// Mitsubishi GX Works2 project: final1   PLC: FX3G

// global labels: Global1
VAR_GLOBAL
  dayOn AT Y000 : BOOL;
  endDay AT M2 : BOOL;
  dayOnn AT X007 : BOOL;
  emergncy AT X005 : BOOL;
  noInventory AT M1 : BOOL;
  dayBegin AT X007 : BOOL;
  sample AT X003 : BOOL;
  analogInput1 AT D8280 : INT;
  realInput AT D1200 : REAL;
END_VAR
VAR_GLOBAL CONSTANT
  const6 : REAL := 6.0;
  const5 : REAL := 5.0;
END_VAR
VAR_GLOBAL
  protein AT M3 : BOOL;
  regular AT M4 : BOOL;
END_VAR
VAR_GLOBAL CONSTANT
  proteinProteinPackageAmount : REAL := 320.0;
  honeytProteinPackageAmount : REAL := 160;
END_VAR
VAR_GLOBAL
  validProtein AT M31 : BOOL;
END_VAR
VAR_GLOBAL CONSTANT
  oatRegularPackageAmount : REAL := 400.0;
  proteinRegularPackageAmount : REAL := 160;
  honeyRegularPackageAmount : REAL := 120;
  honeyProteinPackageAmount : REAL := 160;
END_VAR
VAR_GLOBAL
  validRegular AT M41 : BOOL;
  mixTimer AT TC1 : BOOL;
END_VAR
VAR_GLOBAL CONSTANT
  const50 : INT := 50;
END_VAR
VAR_GLOBAL
  mixTimerOn AT TS1 : BOOL;
  MixLight AT Y003 : BOOL;
  try AT M20 : BOOL;
  oatContain AT D1300 : REAL;
  oatInput AT D1510 : REAL;
  honeyInput AT D1530 : REAL;
  honeyContein AT D1500 : REAL;
  proteinInput AT D1520 : REAL;
  proteinContein AT D1400 : REAL;
END_VAR
VAR_GLOBAL CONSTANT
  oatProteinPackageAmount : REAL := 240.0;
END_VAR
VAR_GLOBAL
  baking AT X002 : BOOL;
  bakeTimerRegular AT TC3 : BOOL;
  bakeTimerProtein AT TC2 : BOOL;
END_VAR
VAR_GLOBAL CONSTANT
  const40 : INT := 40;
END_VAR
VAR_GLOBAL
  bakeTimerProteinON AT TS2 : BOOL;
  bakeTimerRegularON AT TS3 : BOOL;
  flickerHelp AT M6 : BOOL;
  flicker1 AT TC4 : BOOL;
END_VAR
VAR_GLOBAL CONSTANT
  const10 : INT := 10;
END_VAR
VAR_GLOBAL
  flicerTimer1 AT TS4 : BOOL;
  flickerLight1 AT Y001 : BOOL;
  flicker2 AT TC5 : BOOL;
  flicerTimer2 AT TS5 : BOOL;
  flickerLight2 AT Y002 : BOOL;
  finishBake AT M5 : BOOL;
  packing AT X006 : BOOL;
  packingOneBar AT X000 : BOOL;
  countingOneBar AT CC0 : BOOL;
END_VAR
VAR_GLOBAL CONSTANT
  cont1 : INT := 1;
END_VAR
VAR_GLOBAL
  counting8bars AT CC1 : BOOL;
END_VAR
VAR_GLOBAL CONSTANT
  const8 : INT := 8;
END_VAR
VAR_GLOBAL
  counterStarter AT CS0 : BOOL;
  counterStopper AT CS1 : BOOL;
  packingLight AT Y004 : BOOL;
  packageFinished AT M7 : BOOL;
  logInput AT D1250 : REAL;
END_VAR
VAR_GLOBAL CONSTANT
  const400 : REAL := 400.0;
END_VAR
VAR_GLOBAL
  analogPackages AT D1260 : REAL;
  packegesOutput AT D8282 : INT;
END_VAR
VAR_GLOBAL CONSTANT
  const0 : REAL;
  const1 : REAL := 1.0;
END_VAR
VAR_GLOBAL
  totalPackeges AT D1600 : REAL;
  restartPackingCount AT CN1 : INT;
END_VAR
VAR_GLOBAL CONSTANT
  const40Float : REAL := 40.0;
END_VAR
VAR_GLOBAL
  test111 AT M99 : BOOL;
  test888 AT M99 : BOOL;
  noInventory2 AT M19 : BOOL;
END_VAR

// task Task_01 (event TRUE, interval 0, priority 31): POU_01

PROGRAM POU_01
(* structured ladder/FBD written out as ST: instructions are called as NAME(EN, inputs, outputs); _pN, _eN, _tN stand for wires *)
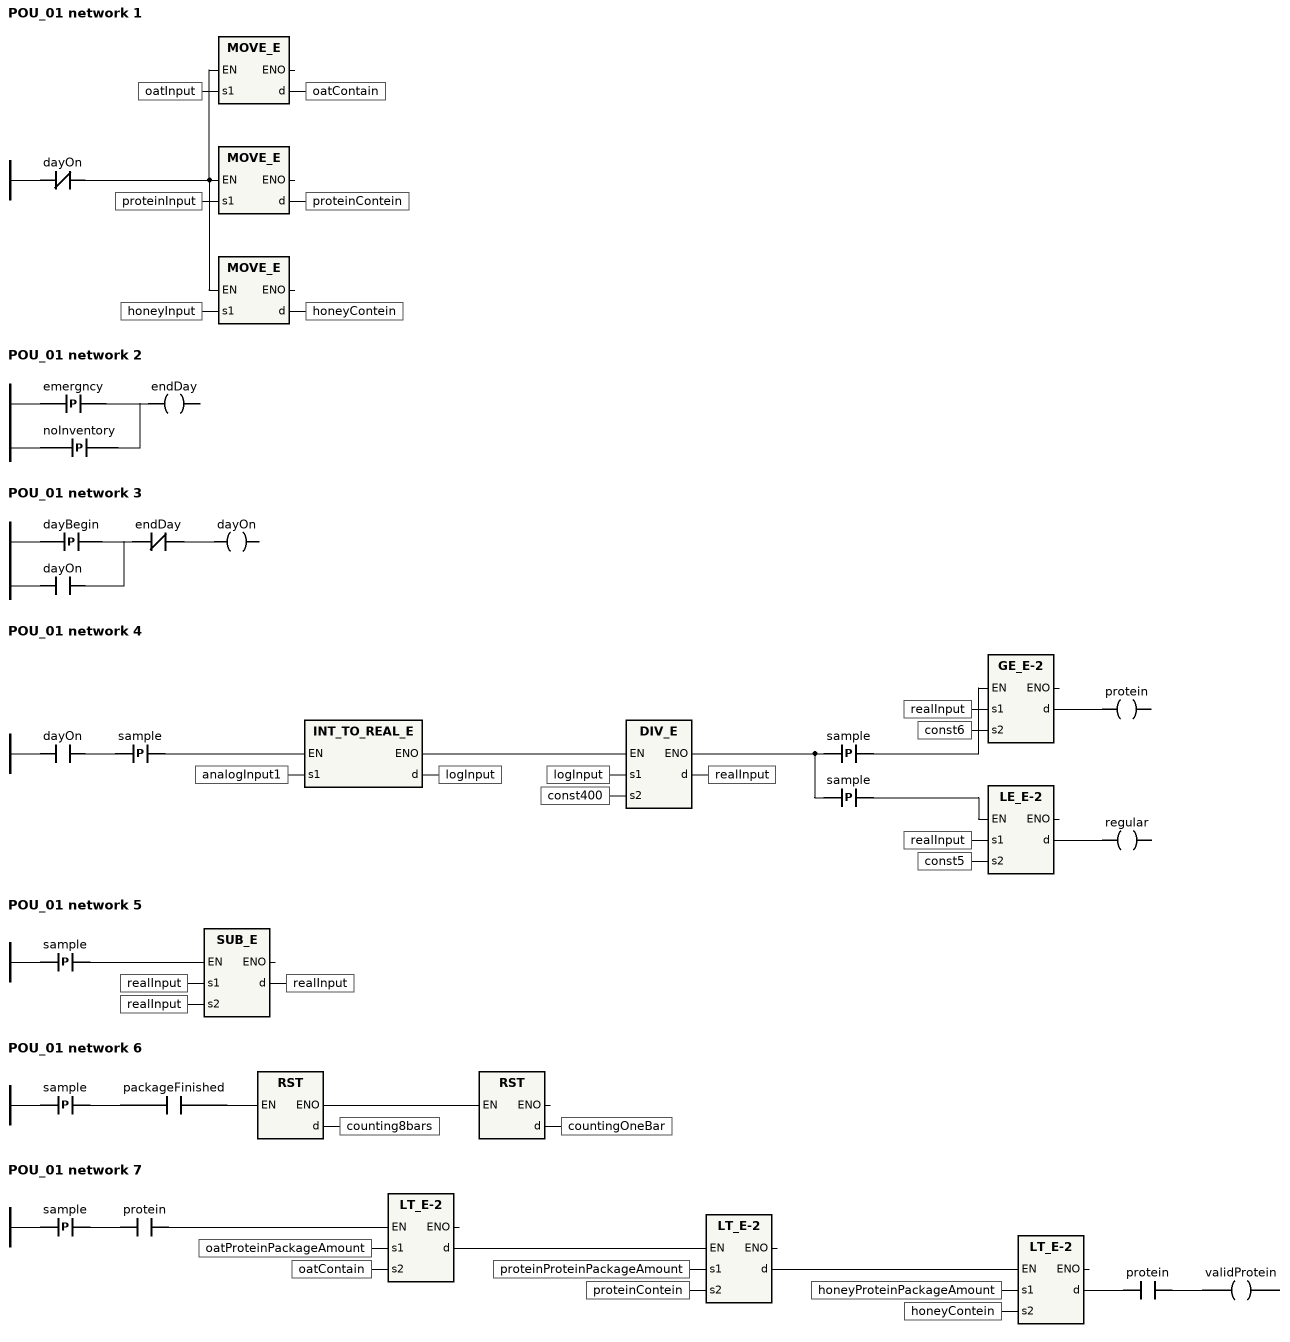
(* network 1 *)
_p1 := NOT dayOn;
MOVE_E(_p1, oatInput, oatContain);
MOVE_E(_p1, proteinInput, proteinContein);
MOVE_E(_p1, honeyInput, honeyContein);
(* network 2 *)
endDay := LDP(TRUE, emergncy) OR LDP(TRUE, noInventory);
(* network 3 *)
dayOn := (LDP(TRUE, dayBegin) OR dayOn) AND NOT endDay;
(* network 4 *)
_e1 := INT_TO_REAL_E(dayOn AND LDP(TRUE, sample), analogInput1, logInput);
_e2 := DIV_E(_e1, logInput, const400, realInput);
GE_E(_e2 AND LDP(TRUE, sample), realInput, const6, _t3);
protein := _t3;
LE_E(_e2 AND LDP(TRUE, sample), realInput, const5, _t4);
regular := _t4;
(* network 5 *)
SUB_E(LDP(TRUE, sample), realInput, realInput, realInput);
(* network 6 *)
_e1 := RST(LDP(TRUE, sample) AND packageFinished, counting8bars);
RST(_e1, countingOneBar);
(* network 7 *)
LT_E(LDP(TRUE, sample) AND protein, oatProteinPackageAmount, oatContain, _t1);
LT_E(_t1, proteinProteinPackageAmount, proteinContein, _t2);
LT_E(_t2, honeyProteinPackageAmount, honeyContein, _t3);
validProtein := _t3 AND protein;
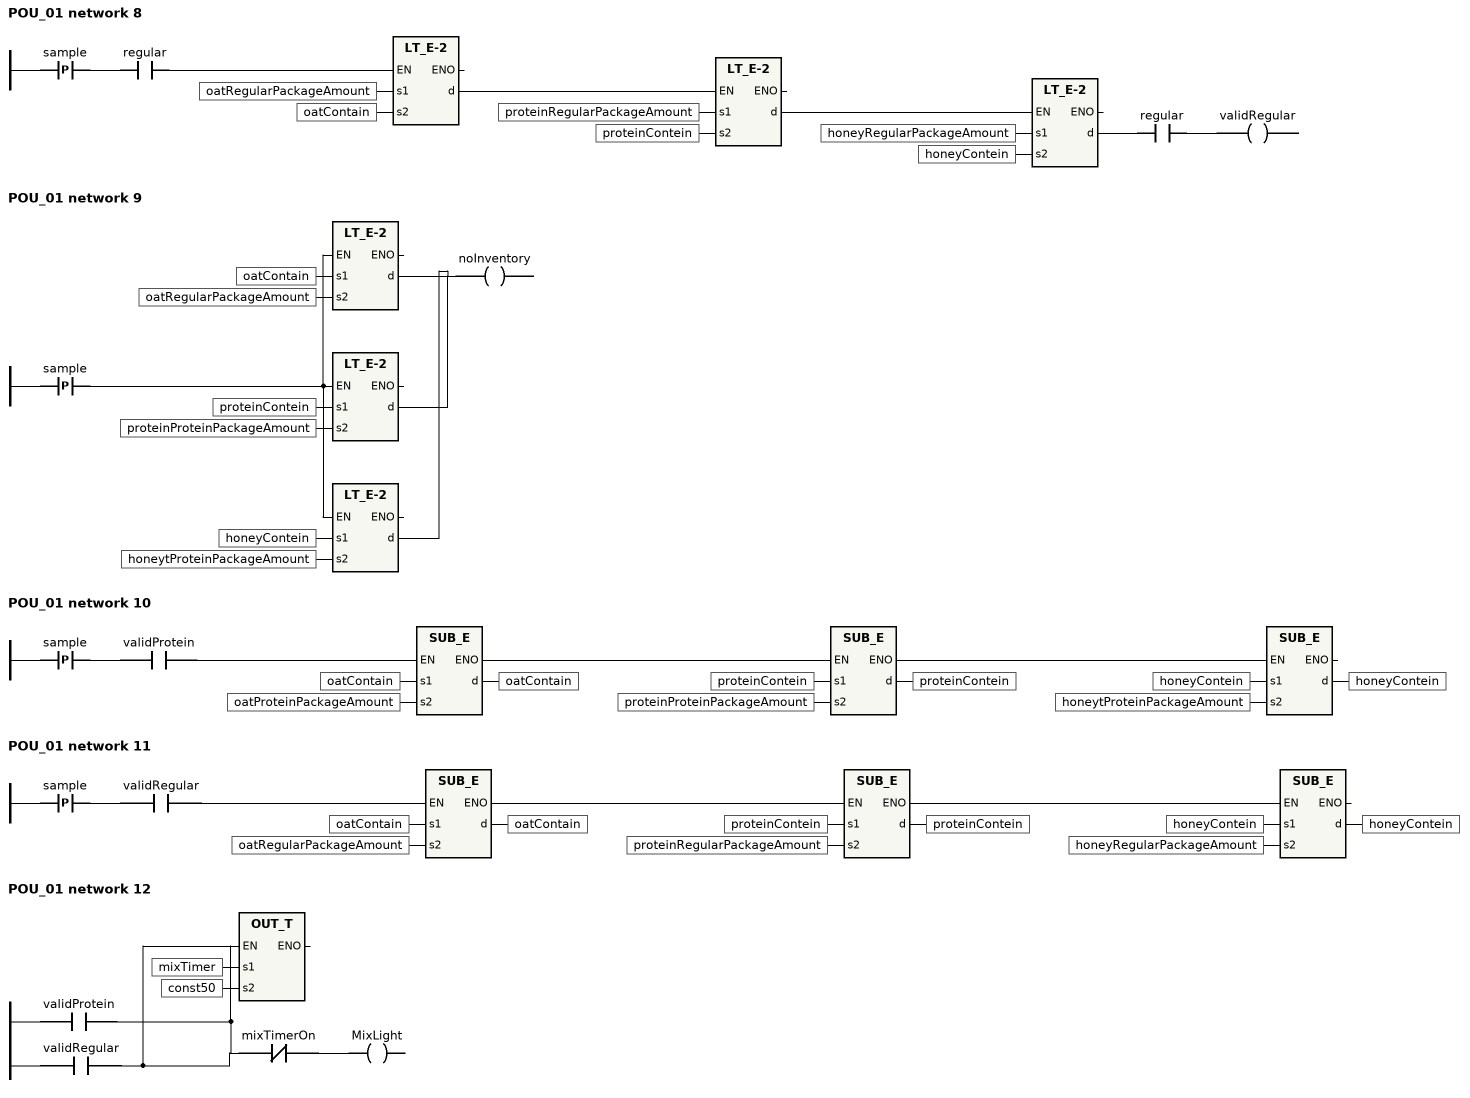
(* network 8 *)
LT_E(LDP(TRUE, sample) AND regular, oatRegularPackageAmount, oatContain, _t1);
LT_E(_t1, proteinRegularPackageAmount, proteinContein, _t2);
LT_E(_t2, honeyRegularPackageAmount, honeyContein, _t3);
validRegular := _t3 AND regular;
(* network 9 *)
_p1 := LDP(TRUE, sample);
LT_E(_p1, oatContain, oatRegularPackageAmount, _t2);
LT_E(_p1, proteinContein, proteinProteinPackageAmount, _t3);
LT_E(_p1, honeyContein, honeytProteinPackageAmount, _t4);
noInventory := _t2 OR _t3 OR _t4;
(* network 10 *)
_e1 := SUB_E(LDP(TRUE, sample) AND validProtein, oatContain, oatProteinPackageAmount, oatContain);
_e2 := SUB_E(_e1, proteinContein, proteinProteinPackageAmount, proteinContein);
SUB_E(_e2, honeyContein, honeytProteinPackageAmount, honeyContein);
(* network 11 *)
_e1 := SUB_E(LDP(TRUE, sample) AND validRegular, oatContain, oatRegularPackageAmount, oatContain);
_e2 := SUB_E(_e1, proteinContein, proteinRegularPackageAmount, proteinContein);
SUB_E(_e2, honeyContein, honeyRegularPackageAmount, honeyContein);
(* network 12 *)
_p1 := validProtein OR validRegular;
OUT_T(_p1, mixTimer, const50);
MixLight := _p1 AND NOT mixTimerOn;
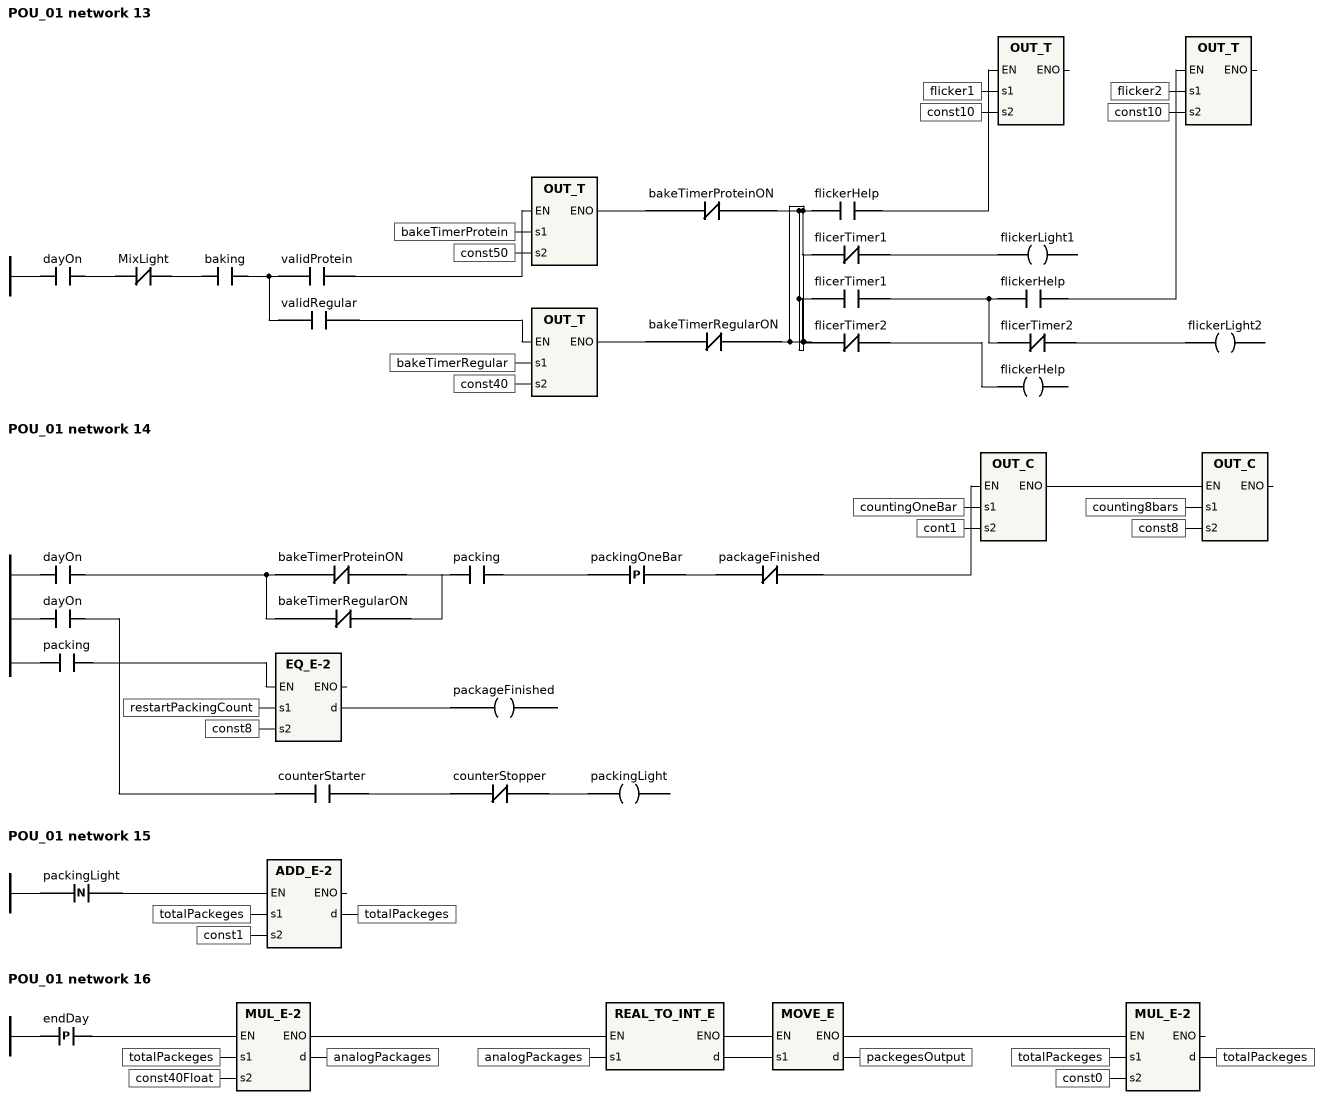
(* network 13 *)
_p1 := dayOn AND NOT MixLight AND baking;
_e2 := OUT_T(_p1 AND validProtein, bakeTimerProtein, const50);
_e3 := OUT_T(_p1 AND validRegular, bakeTimerRegular, const40);
_p4 := (_e2 AND NOT bakeTimerProteinON) OR (_e3 AND NOT bakeTimerRegularON);
OUT_T(_p4 AND flickerHelp, flicker1, const10);
flickerLight1 := _p4 AND NOT flicerTimer1;
_p5 := _p4 AND flicerTimer1;
OUT_T(_p5 AND flickerHelp, flicker2, const10);
flickerLight2 := _p5 AND NOT flicerTimer2;
flickerHelp := _p4 AND NOT flicerTimer2;
(* network 14 *)
_e1 := OUT_C(((((dayOn AND NOT bakeTimerProteinON) OR (dayOn AND NOT bakeTimerRegularON)) AND packing) AND LDP(TRUE, packingOneBar)) AND NOT packageFinished, countingOneBar, cont1);
OUT_C(_e1, counting8bars, const8);
packingLight := dayOn AND counterStarter AND NOT counterStopper;
EQ_E(packing, restartPackingCount, const8, _t2);
packageFinished := _t2;
(* network 15 *)
ADD_E(LDF(TRUE, packingLight), totalPackeges, const1, totalPackeges);
(* network 16 *)
_e1 := MUL_E(LDP(TRUE, endDay), totalPackeges, const40Float, analogPackages);
_e3 := REAL_TO_INT_E(_e1, analogPackages, _t2);
_e4 := MOVE_E(_e3, _t2, packegesOutput);
MUL_E(_e4, totalPackeges, const0, totalPackeges);
END_PROGRAM
